{attribute 'qualified_only'}
{attribute 'strict'}
TYPE DUT :
(
	Aborting := 0,
	Aborted		:= 1,
	
	Clearing	:= 2,
	Stopping	:= 3,
	Stopped		:= 4,
	
	Resetting	:= 5,
	Idle		:= 6,
	Starting	:= 7,
	Execute		:= 8,
	
	Holding		:= 9,
	Held		:= 10,
	Unholding		:= 11,
	
	Suspending		:= 12,
	Suspended		:= 13,
	Unsuspending	:= 14,
	
	Complete 		:= 15
);
END_TYPE

(* stored: Version 1.1.0.1, ProductVersion 3.1.4024.6
   EnumerationTextList DUT: Id {95ed8ca2-9bff-4ecc-b2f3-09146f44728f} *)
